{attribute addProperty Name "LogicCheckerData"}
{attribute 'qlik_value_field:CheckType = Logic'}
TYPE
    TcoDigitalInspectorData EXTENDS TcoInspectorData :
    STRUCT
        (*~
		<docu>
		<summary>
			Required status for the check to Pass.	
		</summary>
		</docu>
	~*)
        {attribute addProperty Name "<#REQUIRED STATUS#>"}
        {attribute 'qlik_load:RequiredStatus'}
        RequiredStatus : BOOL;

        (*~
		<docu>
		<summary>
			Detected status.	
		</summary>
		</docu>
	~*)
        {attribute addProperty Name "<#DETECTED STATUS#>"}
        {attribute clr [RenderIgnore("Control", "ShadowControl")]}
        {attribute 'qlik_load:DetectedStatus'}
        DetectedStatus : BOOL;
    END_STRUCT
END_TYPE

(* stored: Version 1.1.0.1, ProductVersion 3.1.4024.9
   DUT TcoDigitalInspectorData: Id {cd575c1e-dcb1-0a06-301a-c160533158aa} *)
